KUKA KRL program: SOFTINZ.src

&ACCESS RVO1
&REL 52
&PARAM TEMPLATE = C:\KRC\Roboter\Template\FunctionVorgabe
&PARAM EDITMASK = *
DEFFCT BOOL SOFTINZ( )

DECL STIFFNESS USERSTIFF

USERSTIFF=$STIFFNESS
USERSTIFF.STRATEGY=20
USERSTIFF.FRAMETYPE=#TOOL
USERSTIFF.TOOL={X 0.0,Y 0.0,Z 180.0,A 0.0,B 0.0,C 0.0}
USERSTIFF.TOOL=TOOL_DATA[5]
USERSTIFF.BASE=$BASE
USERSTIFF.CPSTIFFNESS={X 2000.0,Y 2000.0,Z 100.0,A 200.0,B 200.0,C 200.0}
USERSTIFF.CPDAMPING={X 0.7,Y 0.7,Z 1.0,A 0.7,B 0.7,C 0.7}
USERSTIFF.AXISSTIFFNESS={A1 2000.0,A2 2000.0,A3 2000.0,A4 2000.0,A5 2000.0,A6 2000.0,E1 2000.0}
USERSTIFF.AXISDAMPING={A1 0.7,A2 0.7,A3 0.7,A4 0.7,A5 0.7,A6 0.7,E1 0.7}
USERSTIFF.CPMAXDELTA={X 7.0,Y 7.0,Z 500.0,A 2.0,B 2.0,C 2.0}
USERSTIFF.MAXFORCE={X 50.0,Y 50.0,Z 50.0,A 10.0,B 10.0,C 10.0}
USERSTIFF.AXISMAXDELTA={A1 30.0,A2 30.0,A3 30.0,A4 30.0,A5 30.0,A6 10.0,E1 10.0}
USERSTIFF.AXISMAXDELTATRQ={A1 5.0,A2 5.0,A3 5.0,A4 5.0,A5 5.0,A6 5.0,E1 5.0}
$STIFFNESS=USERSTIFF

RETURN TRUE
ENDFCT
